TYPE STATE_1 :
(
	DORMANT,
	EXECUTING,
	DONE,
	INERROR,
	ABORTING,
	ABORTED,
	RESETING 
);
END_TYPE

(* stored: Version 1.1.0.1, ProductVersion 3.1.4024.9
   DUT STATE_1: Id {9f3a652f-ff87-4297-87a0-95f1d9765b00} *)
